FUNCTION_BLOCK fb_sv_reset
VAR_IN_OUT
	var_ref_sv : ref_sv_io;
END_VAR
VAR_INPUT
	in_flg_reset : BOOL;
END_VAR
VAR_OUTPUT
	out_flg_resetDone: BOOL;
END_VAR
VAR

	var_process: INT;
	fbi_ton1: TON;
END_VAR


fbi_ton1(IN:= , PT:=T#100MS , Q=> , ET=> );

IF NOT in_flg_reset THEN
	var_process := 0;
END_IF
CASE var_process OF
	0:
		IF in_flg_reset THEN
			fbi_ton1.IN := FALSE;
			var_process := 1;
		END_IF
	1:	
		fbi_ton1.IN := TRUE;
		var_ref_sv.out.out_flg_svA := FALSE;
		var_ref_sv.out.out_flg_svB := FALSE;
		var_ref_sv.param.var_mutex := 0;
		IF fbi_ton1.Q THEN
			var_process := 2;
		END_IF
	2:
		out_flg_resetDone := TRUE;
		var_process := 3;
	3:
		out_flg_resetDone := FALSE;
END_CASE

END_FUNCTION_BLOCK

(* stored: Version 1.1.0.1, ProductVersion 3.1.4024.11
   POU fb_sv_reset: Id {8b56c82f-ef07-4dcc-baea-ae7ef43bc013}, SpecialFunc None *)
